FUNCTION_BLOCK FB_TimeAverage
VAR_INPUT
	IN:		REAL;
	PT:		TIME := T#4400MS;
END_VAR
VAR_OUTPUT
	AVG:	REAL;
	MINAVG:	REAL;
	MAXAVG:	REAL;
	Overflow: BOOL;
END_VAR
VAR
	fbCycle	:TON;
	buffer:	ARRAY[0..30000] OF REAL;
	index:	INT := 0;
	number:	INT := 0;
	i:		INT;
	sum:	REAL;
END_VAR

fbCycle(IN:= NOT fbCycle.Q,
		PT:= PT);

// write the current value into the buffer		
buffer[index] := IN;

// increase the index
IF index < 30000 THEN
	index := index + 1;
END_IF

Overflow := (index = 30000);

// during the first cycle number will be smaller than index
IF number < index THEN
	number := index;
END_IF

// sum up the buffer to the current number
sum := 0.0;
MINAVG := IN;
MAXAVG := IN;
FOR i :=0 TO number-1 DO
	sum := sum + buffer[i];
	MINAVG := MIN(buffer[i], MINAVG);
	MAXAVG := MAX(buffer[i], MAXAVG);
END_FOR

// return the average
AVG := sum / number;

// if we hit the cycle time, reset the index and overwrite old values
IF fbCycle.Q THEN
	number := index;
	index := 0;
END_IF

END_FUNCTION_BLOCK

(* stored: Version 1.1.0.1, ProductVersion 3.1.4024.9
   POU FB_TimeAverage: Id {3d3f768c-9845-48d2-a29c-b1ee2e4a39dc}, SpecialFunc None *)
